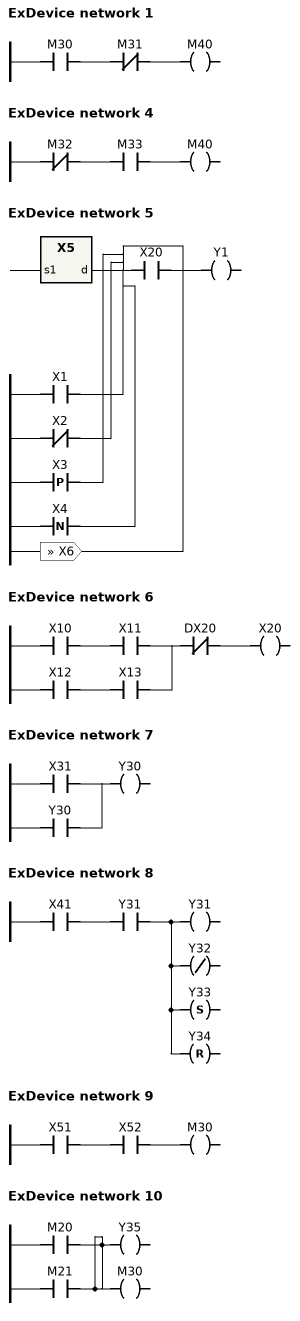
(* network 1 *)
M40 := M30 AND NOT M31;
(* network 4 *)
M40 := NOT M32 AND M33;
(* network 5 *)
(* element kind 19 X5 <- TRUE *)
IF TRUE THEN JMP X6; END_IF;
Y1 := (X1 OR (NOT X2) OR LDP(TRUE, X3) OR LDF(TRUE, X4) OR _feedback OR _feedback) AND X20;
(* network 6 *)
X20 := ((X10 AND X11) OR (X12 AND X13)) AND NOT DX20;
(* network 7 *)
Y30 := X31 OR Y30;
(* network 8 *)
_p1 := X41 AND Y31;
Y31 := _p1;
Y32 := NOT _p1;
SET(_p1, Y33);
RST(_p1, Y34);
(* network 9 *)
M30 := X51 AND X52;
(* network 10 *)
_p1 := M20 OR M21;
Y35 := _p1;
M30 := _p1;
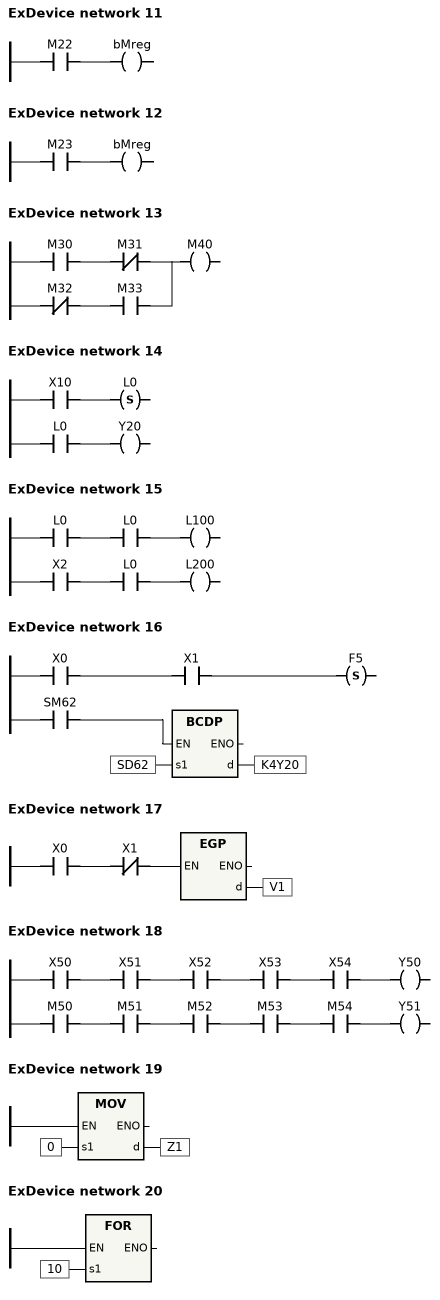
(* network 11 *)
bMreg := M22;
(* network 12 *)
bMreg := M23;
(* network 13 *)
M40 := (M30 AND NOT M31) OR (NOT M32 AND M33);
(* network 14 *)
SET(X10, L0);
Y20 := L0;
(* network 15 *)
L100 := L0 AND L0;
L200 := X2 AND L0;
(* network 16 *)
SET(X0 AND X1, F5);
BCDP(SM62, SD62, K4Y20);
(* network 17 *)
EGP(X0 AND NOT X1, V1);
(* network 18 *)
Y50 := X50 AND X51 AND X52 AND X53 AND X54;
Y51 := M50 AND M51 AND M52 AND M53 AND M54;
(* network 19 *)
MOV(TRUE, 0, Z1);
(* network 20 *)
FOR(TRUE, 10);
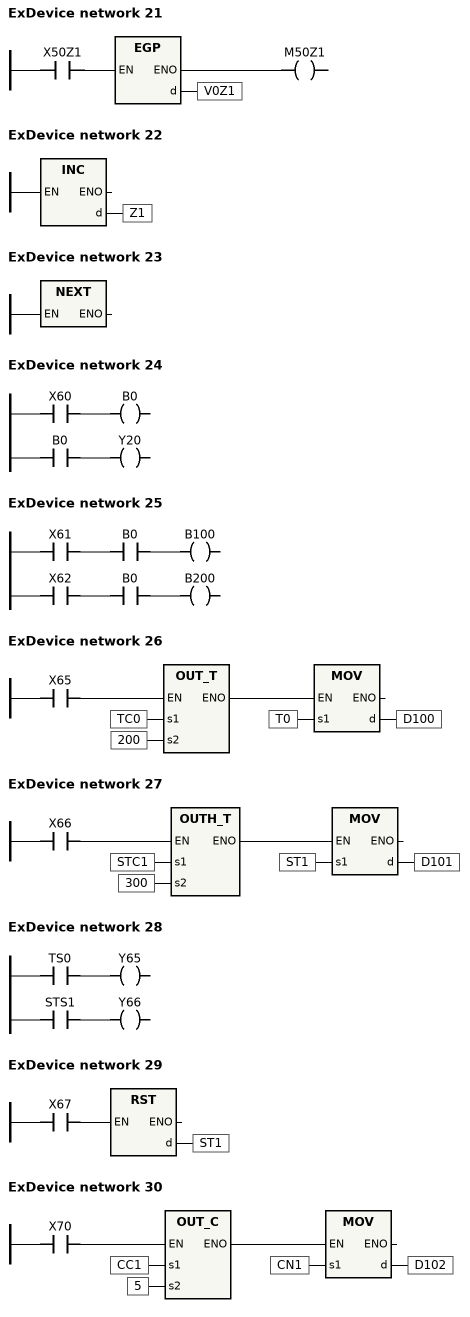
(* network 21 *)
_e1 := EGP(X50Z1, V0Z1);
M50Z1 := _e1;
(* network 22 *)
INC(TRUE, Z1);
(* network 23 *)
NEXT(TRUE);
(* network 24 *)
B0 := X60;
Y20 := B0;
(* network 25 *)
B100 := X61 AND B0;
B200 := X62 AND B0;
(* network 26 *)
_e1 := OUT_T(X65, TC0, 200);
MOV(_e1, T0, D100);
(* network 27 *)
_e1 := OUTH_T(X66, STC1, 300);
MOV(_e1, ST1, D101);
(* network 28 *)
Y65 := TS0;
Y66 := STS1;
(* network 29 *)
RST(X67, ST1);
(* network 30 *)
_e1 := OUT_C(X70, CC1, 5);
MOV(_e1, CN1, D102);
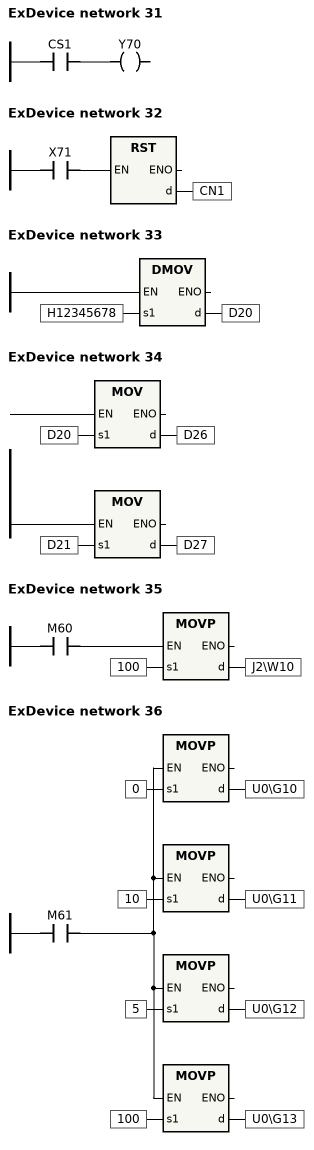
(* network 31 *)
Y70 := CS1;
(* network 32 *)
RST(X71, CN1);
(* network 33 *)
DMOV(TRUE, H12345678, D20);
(* network 34 *)
MOV(TRUE, D20, D26);
MOV(TRUE, D21, D27);
(* network 35 *)
MOVP(M60, 100, J2\W10);
(* network 36 *)
MOVP(M61, 0, U0\G10);
MOVP(M61, 10, U0\G11);
MOVP(M61, 5, U0\G12);
MOVP(M61, 100, U0\G13);
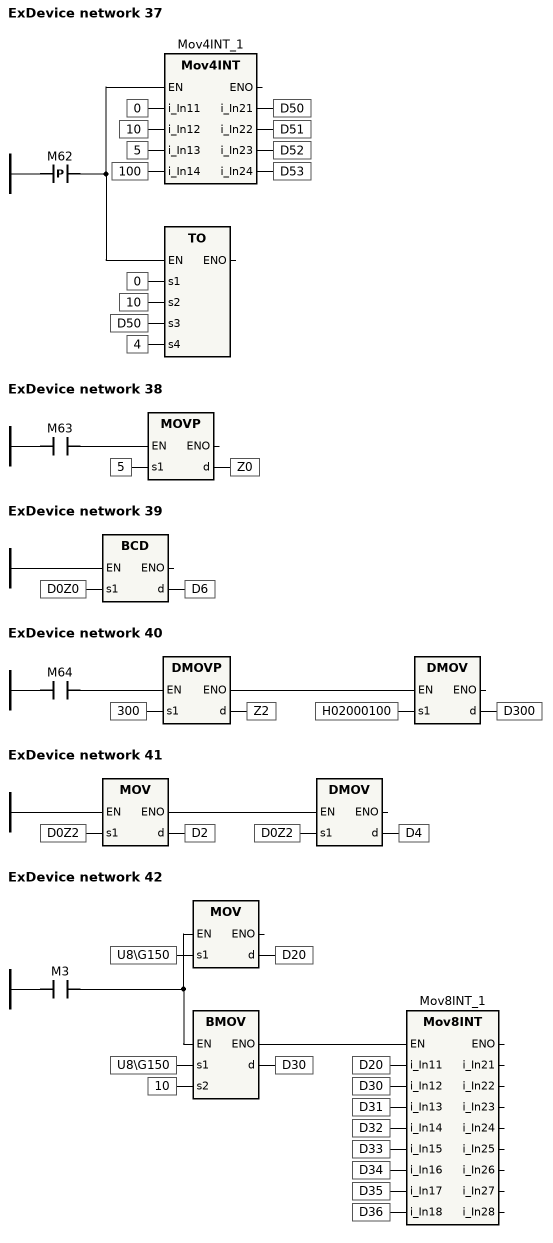
(* network 37 *)
_p1 := LDP(TRUE, M62);
Mov4INT_1(EN := _p1, i_In11 := 0, i_In12 := 10, i_In13 := 5, i_In14 := 100, i_In21 => D50, i_In22 => D51, i_In23 => D52, i_In24 => D53);
TO(_p1, 0, 10, D50, 4);
(* network 38 *)
MOVP(M63, 5, Z0);
(* network 39 *)
BCD(TRUE, D0Z0, D6);
(* network 40 *)
_e1 := DMOVP(M64, 300, Z2);
DMOV(_e1, H02000100, D300);
(* network 41 *)
_e1 := MOV(TRUE, D0Z2, D2);
DMOV(_e1, D0Z2, D4);
(* network 42 *)
MOV(M3, U8\G150, D20);
_e1 := BMOV(M3, U8\G150, 10, D30);
Mov8INT_1(EN := _e1, i_In11 := D20, i_In12 := D30, i_In13 := D31, i_In14 := D32, i_In15 := D33, i_In16 := D34, i_In17 := D35, i_In18 := D36);
END_PROGRAM

PROGRAM ExDouble
(* structured ladder/FBD written out as ST: instructions are called as NAME(EN, inputs, outputs); _pN, _eN, _tN stand for wires *)
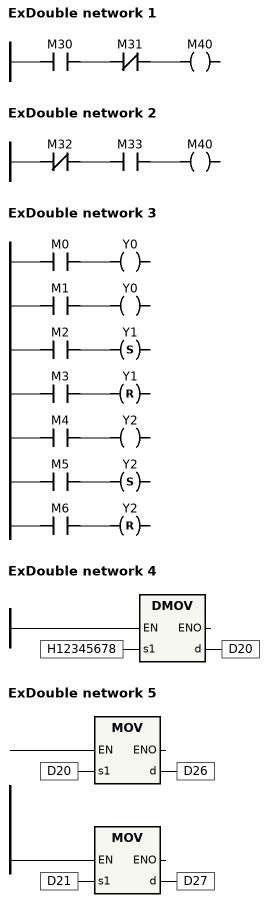
(* network 1 *)
M40 := M30 AND NOT M31;
(* network 2 *)
M40 := NOT M32 AND M33;
(* network 3 *)
Y0 := M0;
Y0 := M1;
SET(M2, Y1);
RST(M3, Y1);
Y2 := M4;
SET(M5, Y2);
RST(M6, Y2);
(* network 4 *)
DMOV(TRUE, H12345678, D20);
(* network 5 *)
MOV(TRUE, D20, D26);
MOV(TRUE, D21, D27);
END_PROGRAM

PROGRAM ExIndex
VAR
  GetInt : INT;
  NthBit : INT;
  SetInt : INT;
  SetInt2 : INT;
  giArea : ARRAY [0..99] OF INT;
  gdPos : ARRAY [0..99] OF DINT;
END_VAR
(* structured ladder/FBD written out as ST: instructions are called as NAME(EN, inputs, outputs); _pN, _eN, _tN stand for wires *)
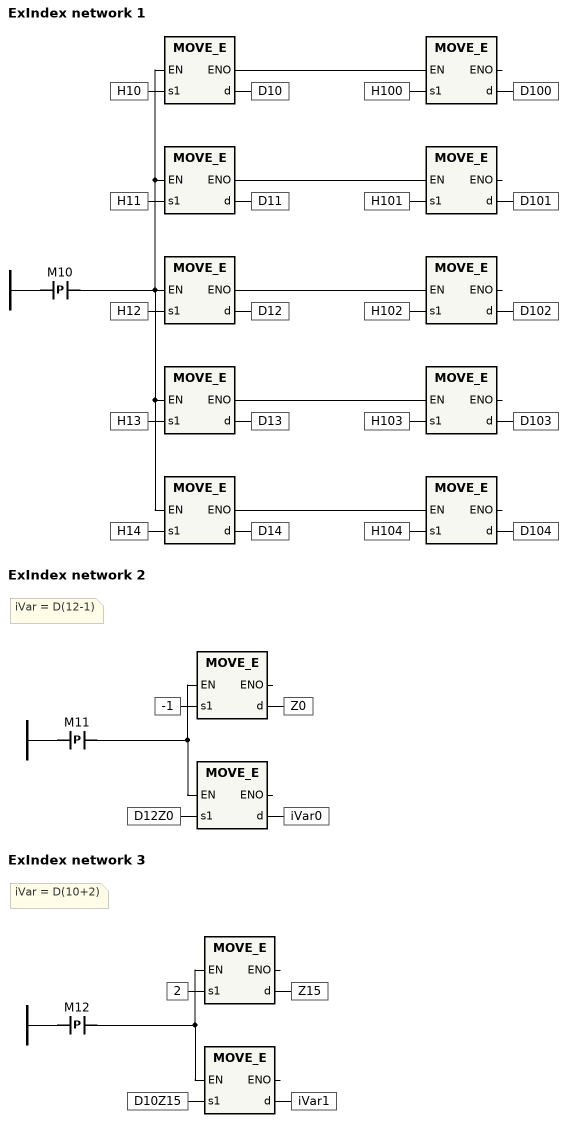
(* network 1 *)
_p1 := LDP(TRUE, M10);
_e2 := MOVE_E(_p1, H10, D10);
MOVE_E(_e2, H100, D100);
_e3 := MOVE_E(_p1, H11, D11);
MOVE_E(_e3, H101, D101);
_e4 := MOVE_E(_p1, H12, D12);
MOVE_E(_e4, H102, D102);
_e5 := MOVE_E(_p1, H13, D13);
MOVE_E(_e5, H103, D103);
_e6 := MOVE_E(_p1, H14, D14);
MOVE_E(_e6, H104, D104);
(* network 2 *)
(* iVar = D(12-1) *)
_p1 := LDP(TRUE, M11);
MOVE_E(_p1, -1, Z0);
MOVE_E(_p1, D12Z0, iVar0);
(* network 3 *)
(* iVar = D(10+2) *)
_p1 := LDP(TRUE, M12);
MOVE_E(_p1, 2, Z15);
MOVE_E(_p1, D10Z15, iVar1);
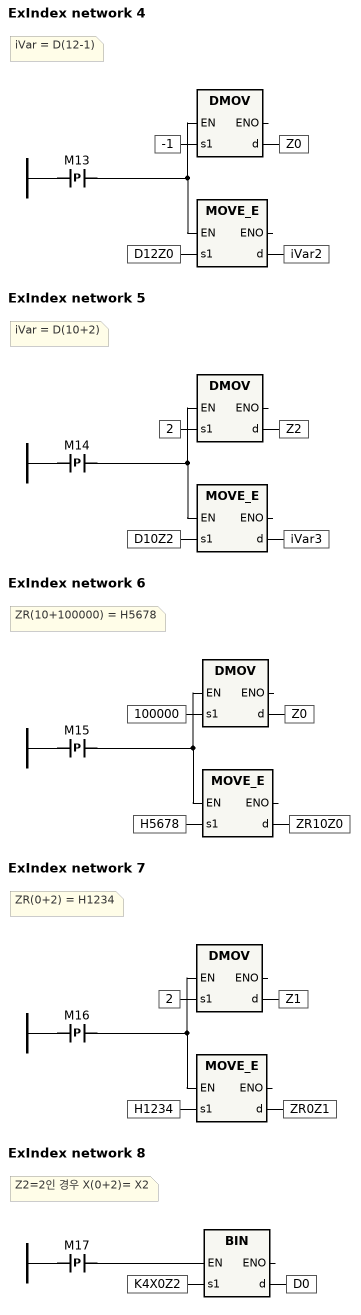
(* network 4 *)
(* iVar = D(12-1) *)
_p1 := LDP(TRUE, M13);
DMOV(_p1, -1, Z0);
MOVE_E(_p1, D12Z0, iVar2);
(* network 5 *)
(* iVar = D(10+2) *)
_p1 := LDP(TRUE, M14);
DMOV(_p1, 2, Z2);
MOVE_E(_p1, D10Z2, iVar3);
(* network 6 *)
(* ZR(10+100000) = H5678 *)
_p1 := LDP(TRUE, M15);
DMOV(_p1, 100000, Z0);
MOVE_E(_p1, H5678, ZR10Z0);
(* network 7 *)
(* ZR(0+2) = H1234 *)
_p1 := LDP(TRUE, M16);
DMOV(_p1, 2, Z1);
MOVE_E(_p1, H1234, ZR0Z1);
(* network 8 *)
(* Z2=2인 경우 X(0+2)= X2 *)
BIN(LDP(TRUE, M17), K4X0Z2, D0);
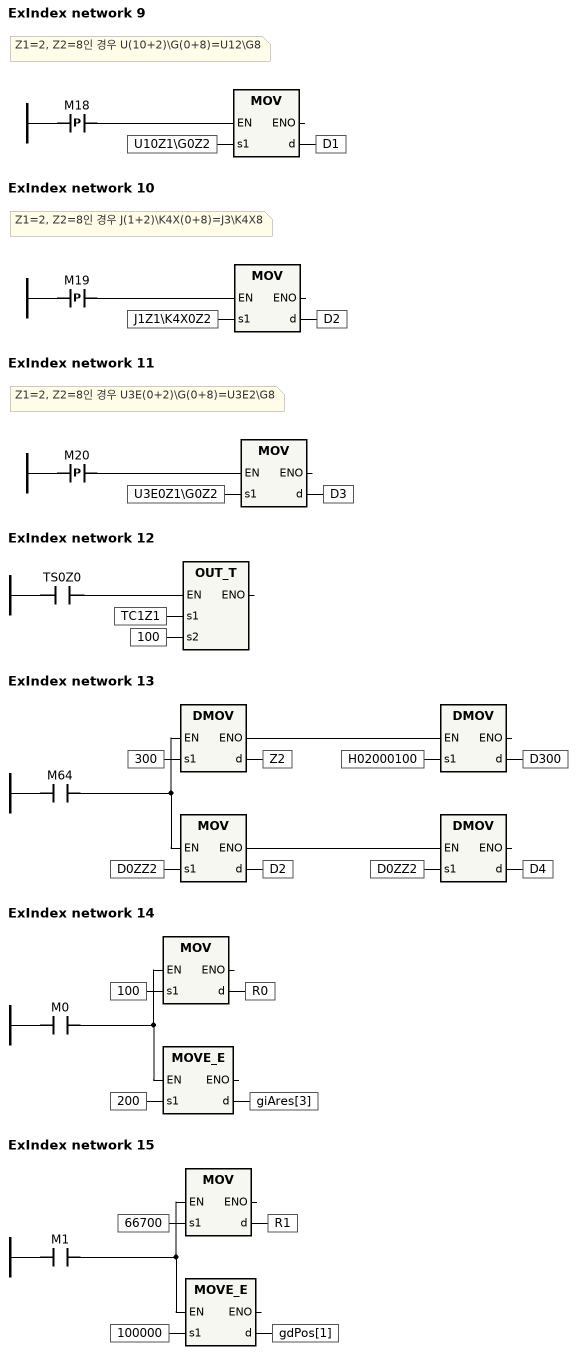
(* network 9 *)
(* Z1=2, Z2=8인 경우 U(10+2)\G(0+8)=U12\G8 *)
MOV(LDP(TRUE, M18), U10Z1\G0Z2, D1);
(* network 10 *)
(* Z1=2, Z2=8인 경우 J(1+2)\K4X(0+8)=J3\K4X8 *)
MOV(LDP(TRUE, M19), J1Z1\K4X0Z2, D2);
(* network 11 *)
(* Z1=2, Z2=8인 경우 U3E(0+2)\G(0+8)=U3E2\G8 *)
MOV(LDP(TRUE, M20), U3E0Z1\G0Z2, D3);
(* network 12 *)
OUT_T(TS0Z0, TC1Z1, 100);
(* network 13 *)
_e1 := DMOV(M64, 300, Z2);
DMOV(_e1, H02000100, D300);
_e2 := MOV(M64, D0ZZ2, D2);
DMOV(_e2, D0ZZ2, D4);
(* network 14 *)
MOV(M0, 100, R0);
MOVE_E(M0, 200, giAres[3]);
(* network 15 *)
MOV(M1, 66700, R1);
MOVE_E(M1, 100000, gdPos[1]);
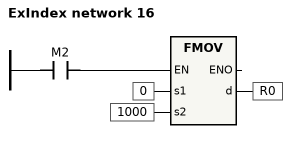
(* network 16 *)
FMOV(M2, 0, 1000, R0);
END_PROGRAM

PROGRAM ExDeviceX
(* structured ladder/FBD written out as ST: instructions are called as NAME(EN, inputs, outputs); _pN, _eN, _tN stand for wires *)
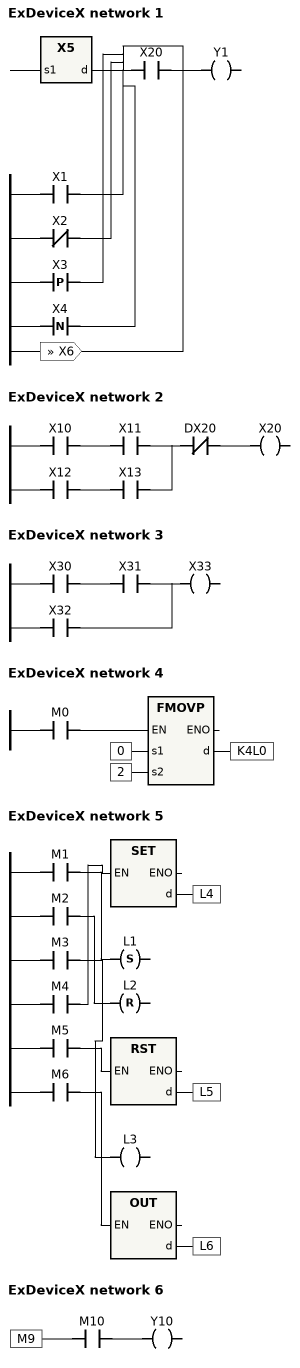
(* network 1 *)
(* element kind 19 X5 <- TRUE *)
IF TRUE THEN JMP X6; END_IF;
Y1 := (X1 OR (NOT X2) OR LDP(TRUE, X3) OR LDF(TRUE, X4) OR _feedback OR _feedback) AND X20;
(* network 2 *)
X20 := ((X10 AND X11) OR (X12 AND X13)) AND NOT DX20;
(* network 3 *)
X33 := (X30 AND X31) OR X32;
(* network 4 *)
FMOVP(M0, 0, 2, K4L0);
(* network 5 *)
SET(M1, L1);
RST(M2, L2);
L3 := M3;
SET(M4, L4);
RST(M5, L5);
OUT(M6, L6);
(* network 6 *)
Y10 := M9 AND M10;
END_PROGRAM

FUNCTION_BLOCK Word2Bit
VAR_INPUT
  IN : WORD;
END_VAR
VAR_OUTPUT
  Bit0 : BOOL;
  Bit1 : BOOL;
  Bit2 : BOOL;
  Bit3 : BOOL;
  Bit4 : BOOL;
  Bit5 : BOOL;
  Bit6 : BOOL;
  Bit7 : BOOL;
  Bit8 : BOOL;
  Bit9 : BOOL;
  Bit10 : BOOL;
  Bit11 : BOOL;
  Bit12 : BOOL;
  Bit13 : BOOL;
  Bit14 : BOOL;
  Bit15 : BOOL;
END_VAR
 
Bit0 := WORD_TO_BOOL(IN AND 16#0001);
Bit1 := WORD_TO_BOOL(SHR(IN AND 16#0002 , 1));
Bit2 := WORD_TO_BOOL(SHR(IN AND 16#0004 , 2));
Bit3 := WORD_TO_BOOL(SHR(IN AND 16#0008 , 3));
Bit4 := WORD_TO_BOOL(SHR(IN AND 16#0010 , 4));
Bit5 := WORD_TO_BOOL(SHR(IN AND 16#0020 , 5));
Bit6 := WORD_TO_BOOL(SHR(IN AND 16#0040 , 6));
Bit7 := WORD_TO_BOOL(SHR(IN AND 16#0080 , 7));
Bit8 := WORD_TO_BOOL(SHR(IN AND 16#0100 , 8));
Bit9 := WORD_TO_BOOL(SHR(IN AND 16#0200 , 9));
Bit10 := WORD_TO_BOOL(SHR(IN AND 16#0400 , 10));
Bit11 := WORD_TO_BOOL(SHR(IN AND 16#0800 , 11));
Bit12 := WORD_TO_BOOL(SHR(IN AND 16#1000 , 12));
Bit13 := WORD_TO_BOOL(SHR(IN AND 16#2000 , 13));
Bit14 := WORD_TO_BOOL(SHR(IN AND 16#4000 , 14));
Bit15 := WORD_TO_BOOL(SHR(IN AND 16#8000 , 15));
END_FUNCTION_BLOCK
